FUNCTION Convert_TIME_TO_BYTE : Hresult
VAR_INPUT
	in : TIME;
	out : REFERENCE TO BYTE;
END_VAR
VAR
	converted : BYTE;
END_VAR

converted := TIME_TO_BYTE(in);

IF (BYTE_TO_TIME(converted) <> in) THEN
	Convert_TIME_TO_BYTE := INCOMPATIBLE;
	RETURN;
END_IF

out := converted;

END_FUNCTION

(* stored: Version 1.1.0.1, ProductVersion 3.1.4024.12
   POU Convert_TIME_TO_BYTE: Id {a04d480a-e328-4f73-aee3-8cc8e8373778}, SpecialFunc None *)
